INTERFACE I_XtsMotorModule

METHOD AcknowledgeMessages : BOOL
VAR_INPUT
END_VAR
END_METHOD

PROPERTY Act24Vdc : LREAL
GET
END_GET
END_PROPERTY

PROPERTY Act48Vdc : LREAL
GET
END_GET
END_PROPERTY

PROPERTY ControlVdcOK : BOOL
GET
END_GET
END_PROPERTY

PROPERTY MotorVdcOK : BOOL
GET
END_GET
END_PROPERTY

METHOD SetInSim : HRESULT
VAR_INPUT
END_VAR
END_METHOD

END_INTERFACE

(* stored: Version 1.1.0.1
   Itf I_XtsMotorModule: Id {3515393f-36cc-43f5-8d97-3f2cabdfbcb7}
   Method AcknowledgeMessages: Id {e3c3ebb1-217b-47ed-9437-e65258d0035f}
   Property Act24Vdc: Id {0d259e55-9237-482e-8220-086e0fe799d4}
   Get Get: Id {c8e0d2e3-2bd9-41e7-8c8b-c44d749a0de0}
   Property Act48Vdc: Id {c9d87ad5-8f23-40fc-a640-b1a3a1673b37}
   Get Get: Id {c4d7bdad-76e1-411d-b065-0aefa174222e}
   Property ControlVdcOK: Id {6dfe739d-2bd0-478b-954e-24f485d24353}
   Get Get: Id {b35844c4-1383-4886-b58f-1632ab1bd8b9}
   Property MotorVdcOK: Id {09e96d28-cf5a-4f0f-9803-ebb77f99ab92}
   Get Get: Id {c580371c-cfa3-490c-912e-33dc7d2b2cc9}
   Method SetInSim: Id {3ed874bb-c6ca-41ec-85c6-4bc2517bd458} *)
